TYPE STM_Control :
STRUCT
	Control : STM_Control_Control;
END_STRUCT
END_TYPE

(* stored: Version 1.1.0.1, ProductVersion 3.1.4024.3
   DUT STM_Control: Id {7fc4b5d8-940c-456f-bf66-83838bd02a14} *)
